// TIA Portal V20 export
DATA_BLOCK "SBK12"   // DB325
// stored: MemoryReserve 100
   VAR
      "ANODE CONVEYOR COVER BACKWARD" : Bool := FALSE;
      "CATHODE CONVEYOR COVER BACKWARD" : Bool := FALSE;
      SPARE : Bool := FALSE;
      SPARE_1 : Bool := FALSE;
      "ANODE CONVEYOR COVER FORWARD" : Bool := FALSE;
      "CATHODE CONVEYOR COVER FORWARD" : Bool := FALSE;
      SPARE_2 : Bool := FALSE;
      SPARE_3 : Bool := FALSE;
      SPARE_4 : Bool;
      SPARE_5 : Bool;
      SPARE_6 : Bool;
   END_VAR
BEGIN
END_DATA_BLOCK
